FUNCTION_BLOCK FB_ADTreatyGauge
VAR_INPUT
END_VAR
VAR_OUTPUT
	{attribute 'pytmc' := '
    pv: 
	'}
	AD_Gauge : ST_VG;
END_VAR
VAR
	//	Setpoint agreed upon w/ AD signified by the signal they send. 
	rTREATY_SIGNAL_PRESS : REAL := 5E-6;
	
	// Presumed pressure if AD's signal is not received. 
	rNO_SIGNAL_PRESS : REAL := 760;
	
	// Input from AD's system indicating pressure belopw setpoint. 
	i_xAD_Press_OK AT %I* : BOOL;
END_VAR

IF i_xAD_Press_OK = TRUE THEN
	AD_Gauge.rPRESS := rTREATY_SIGNAL_PRESS;
	AD_Gauge.xPRESS_OK := TRUE; 
ELSE
	AD_Gauge.rPRESS := rNO_SIGNAL_PRESS;
	AD_Gauge.xPRESS_OK := FALSE; 
END_IF

END_FUNCTION_BLOCK

(* stored: Version 1.1.0.1, ProductVersion 3.1.4024.0
   POU FB_ADTreatyGauge: Id {14900fd8-a061-464a-85fc-d379f9247d46}, SpecialFunc None *)
